{attribute 'linkalways'} 
{attribute 'no_explicit_call' := 'This FB is a CLASS and must be accessed using methods or properties'}
{attribute 'enable_dynamic_creation'}
FUNCTION_BLOCK GlobalInstanceMembers
VAR_STAT // singleton
	instances : InstanceCollection;
	instanceAddedEvent : InstanceAddedEvent;
	instanceRemovedEvent : InstanceRemovedEvent;
END_VAR

METHOD PUBLIC AddInstance
VAR_INPUT
	Instance : I_Instance;
END_VAR
IF Instance = 0 THEN
	RETURN;
END_IF

instances.Insert(Instance);
instanceAddedEvent.Notify(Instance);
END_METHOD

METHOD PUBLIC ForEachInstance
VAR_INPUT
	Visitor : I_VisitIntances;
END_VAR
VAR
	last : DINT;
	i : DINT;
END_VAR
last := instances.Count - 1;

FOR i := 0 TO last DO
	Visitor.Visit(instances.GetByIndex(i));
END_FOR
END_METHOD

PROPERTY PUBLIC OnInstanceAdded : I_Event
GET
OnInstanceAdded := instanceAddedEvent;
END_GET
END_PROPERTY

PROPERTY PUBLIC OnInstanceRemoved : I_Event
GET
OnInstanceRemoved := InstanceRemovedEvent;
END_GET
END_PROPERTY

METHOD PUBLIC RemoveInstance
VAR_INPUT
	Instance : I_Instance;
END_VAR
IF Instance = 0 THEN
	RETURN;
END_IF

instances.Remove(Instance);
InstanceRemovedEvent.Notify(Instance);
END_METHOD

END_FUNCTION_BLOCK

(* stored: Version 1.1.0.1, ProductVersion 3.1.4024.12
   POU GlobalInstanceMembers: Id {d233986c-3a7e-03b5-2e59-ae42bafc7d25}, SpecialFunc None
   Method AddInstance: Id {48e0fdac-0aca-0bda-034e-3a401a41d582}
   Method ForEachInstance: Id {bf191d31-c1c7-0d4d-02f4-17a3ef8b0848}
   Property OnInstanceAdded: Id {600584d7-414e-0905-2bc7-a745ca9d8187}
   Get Get: Id {459c9e98-5661-0a11-2ab3-5eb20ec39307}
   Property OnInstanceRemoved: Id {d08387d4-326d-0c81-1682-6d2d3490dd75}
   Get Get: Id {294daf3c-55c3-05be-17af-48ff32951711}
   Method RemoveInstance: Id {13129834-646e-00fd-0aa3-5528ff194698} *)
